# EPICS substitutions: iocBoot/ioc13bma/auto_shutter.substitutions
file "$(CARS)/CARSApp/Db/auto_shutter.db"
{
pattern
{P,      SHUT, SHUT_STATUS,       SHUT_CONTROL,        PERIOD, BEAM_READY}
{13BMA:, FOE,  13BMA:eps_mbbi4,   13BMA:OpenFEShutter,  30,    PA:13BM:A_BEAM_READY}
{13BMA:, BMC,  13BMA:eps_mbbi100, 13BMA:OpenBMCShutter, 30,    PA:13BM:C_BEAM_READY}
{13BMA:, BMD,  13BMA:eps_mbbi99,  13BMA:OpenBMDShutter, 30,    PA:13BM:D_BEAM_READY}
}
